FUNCTION_BLOCK Turn_Table
VAR_INPUT
END_VAR
VAR_OUTPUT
END_VAR
VAR
END_VAR

// Homing sequence
IF NOT Memory.TurnTableRefDone OR Memory.TurnTableRef THEN
    Memory.TurnTableFwdCmd := TRUE;   // drive forward until reference
    IF IO.TurnTableOutput.o_TurnTable_REF_SENSOR THEN
        Memory.TurnTableFwdCmd := FALSE;
        Memory.TurnTableRefDone := TRUE;   // reference complete
    END_IF;
END_IF;

// Forward rotation
IF Memory.TurnTableFwdCmd AND Memory.TurnTableRefDone THEN
    Memory.TurnTableRev := FALSE;   // interlock
END_IF;

IF IO.TurnTableOutput.o_TurnTable_FWD_SENSOR THEN
    Memory.TurnTableFwd := TRUE;
END_IF;

// Reverse rotation
IF Memory.TurnTableRevCmd AND Memory.TurnTableRefDone THEN
    Memory.TurnTableFwd := FALSE;   // interlock
END_IF;

IF IO.TurnTableOutput.o_TurnTable_REV_SENSOR THEN
    Memory.TurnTableRev := TRUE;
END_IF;

END_FUNCTION_BLOCK

(* stored: Version 1.1.0.1, ProductVersion 3.1.4024.16
   POU Turn_Table: Id {dce6177d-056a-4d74-a031-d1c376a3bb20}, SpecialFunc None *)
